FUNCTION_BLOCK MqttStateFormatter (* Basic FB - INT state to STRING payload for MQTT publish *)
  (* Standard: 61499-2 *)
  (* Version 0.1, 5/22/2026, easensoy, WMG, v1 bare state-to-string *)
  PACKAGE Main;
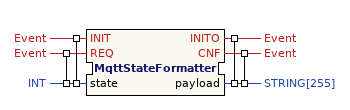
  EVENT_INPUT
    INIT WITH state; (* Initialization Request *)
    REQ WITH state; (* Format on state change *)
  END_EVENT
  EVENT_OUTPUT
    INITO WITH payload; (* Initialization Confirm *)
    CNF WITH payload; (* Payload ready *)
  END_EVENT
  VAR_INPUT
    state : INT; (* current_state_to_process *)
  END_VAR
  VAR_OUTPUT
    payload : STRING[255]; (* MQTT payload (state as text). Sized [255] so EAE does not flag WRN_UNSIZED_STRING (the yellow pin marker) inside every actuator/sensor CAT. *)
  END_VAR
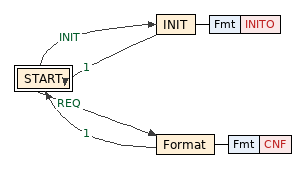
  EC_STATES
    START; (* Initial State *)
    INIT : Fmt -> INITO;
    Format : Fmt -> CNF;
  END_STATES
  EC_TRANSITIONS
    START TO INIT := INIT;
    INIT TO START := 1;
    START TO Format := REQ;
    Format TO START := 1;
  END_TRANSITIONS
  ALGORITHM INIT IN ST: (* Initialization algorithm *)
;
  END_ALGORITHM
  ALGORITHM Fmt IN ST: (* INT state to JSON payload *)
payload := CONCAT(CONCAT('{state:', INT_TO_STRING(state)), '}');
  END_ALGORITHM
END_FUNCTION_BLOCK
